FUNCTION_BLOCK FuseChannelExtended EXTENDS FuseChannelBasic IMPLEMENTS IFuseChannelExtended
VAR_INPUT
END_VAR
VAR_OUTPUT
END_VAR
VAR
	_ChnEx : EL922x_ChannelExtended;
END_VAR


PROPERTY DisabledByDI : BOOL
GET
DisabledByDI := _ChnEx.Status.DisabledByDI;
END_GET
END_PROPERTY


PROPERTY DisabledByOutput : BOOL
GET
DisabledByOutput := _ChnEx.Status.DisabledByOutput;
END_GET
END_PROPERTY


PROPERTY DisabledBySwitch : BOOL
GET
DisabledBySwitch := _ChnEx.Status.DisabledBySwitch;
END_GET
END_PROPERTY


PROPERTY Overload : BOOL
GET
Overload := _ChnEx.Status.Overload;
END_GET
END_PROPERTY


PROPERTY Overvoltage : BOOL
GET
Overvoltage := _ChnEx.Status.Overvoltage;
END_GET
END_PROPERTY

{warning 'add property implementation'}
PROPERTY ShortCircuit : BOOL
GET
ShortCircuit := _ChnEx.Status.ShortCircuit;
END_GET
END_PROPERTY

{warning 'add property implementation'}
PROPERTY StateDeviceSwitch : BOOL
GET
StateDeviceSwitch := _ChnEx.Status.StateDeviceSwitch;
END_GET
END_PROPERTY

{warning 'add property implementation'}
PROPERTY StateDigitalInput : BOOL
GET
StateDigitalInput := _ChnEx.Status.StateDigitalInput;
END_GET
END_PROPERTY

{warning 'add property implementation'}
PROPERTY Undervoltage : BOOL
GET
Undervoltage := _ChnEx.Status.Undervoltage;
END_GET
END_PROPERTY

END_FUNCTION_BLOCK

(* stored: Version 1.1.0.1, ProductVersion 3.1.4024.6
   POU FuseChannelExtended: Id {9757487c-991c-4df2-9a74-8898cc78a011}, SpecialFunc None
   Property DisabledByDI: Id {2150f53c-023b-4828-bdb2-98cb9d13e37e}
   Get Get: Id {d51d9500-f825-47d9-819d-b13e41232920}
   Property DisabledByOutput: Id {49f0e1d6-d31a-4a95-a0b1-f022ee3c0537}
   Get Get: Id {beed161c-dbe7-4ef4-8576-41104c020510}
   Property DisabledBySwitch: Id {1a824d32-5cc9-491e-a5e2-e068b8d7adc3}
   Get Get: Id {d0922947-56fe-4875-a8b3-28f631092c80}
   Property Overload: Id {347322a6-d7e5-4ecc-bd2c-eae47d597746}
   Get Get: Id {0c479487-50e2-41b4-b043-ded7d4bd097a}
   Property Overvoltage: Id {e4a6bc9a-5932-44c2-bb0f-76e22b4abdd1}
   Get Get: Id {8647ee9c-f952-46d5-8d97-330b212329ab}
   Property ShortCircuit: Id {9ce84636-7137-4650-bbb7-ef74246b3894}
   Get Get: Id {e012670f-9951-4635-ac0d-f2a05774f78b}
   Property StateDeviceSwitch: Id {295930d7-b796-41d9-90dd-2bb675c52ebc}
   Get Get: Id {e5986a7f-4804-491d-9696-f6f973680fb0}
   Property StateDigitalInput: Id {7180d8b0-db95-4cb6-98a7-266b9368556a}
   Get Get: Id {7f2fdffc-4b5a-480e-9b45-27af82e8831a}
   Property Undervoltage: Id {0a5421cf-8f28-4525-8a8c-a201222b869b}
   Get Get: Id {038e1e13-0cf5-44d3-ab0d-f736da527dc1} *)
